(* Logix 5000 project; controller code_tcc vendor 1 type 14 code 106 rev 33.11; software revision 33.01; part 3 of 3 *)
(* tags used below, declared in another part *)
   Count : INT;
   Wrk_TransactionPtr : DINT;
(* raC_Tec_NetModbusTCPClient_ChkWrReply, continued *)

ROUTINE Prescan   (* ladder *)
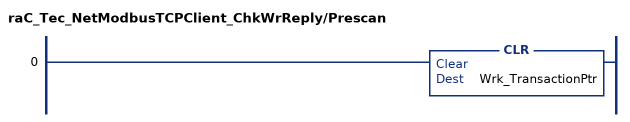
   0: CLR(Wrk_TransactionPtr);
END_ROUTINE
END_ADD_ON_INSTRUCTION

ADD_ON_INSTRUCTION raC_Tec_NetModbusTCPClient_RespStrBit   (* revision 2.0, ExecutePrescan *)
VAR_INPUT
   Inputs : BOOL; {required}
   Modbus_CMD_Len : INT; {required}
   LocalOffset : INT; {required}
END_VAR
VAR_IN_OUT
   ModbusData : raC_UDT_ModbusClientData; {required}
   CommandString : STR0500; {required}
END_VAR
VAR
   Wrk_BufferByteIndex : DINT; {access None}
   Wrk_Cmd_Last : INT; {access None}
   Wrk_Index : DINT; {access None}
   Wrk_BufferBitIndex : DINT; {access None}
   Wrk_ArraySize : DINT; {access None}
END_VAR

ROUTINE Logic   (* ladder *)
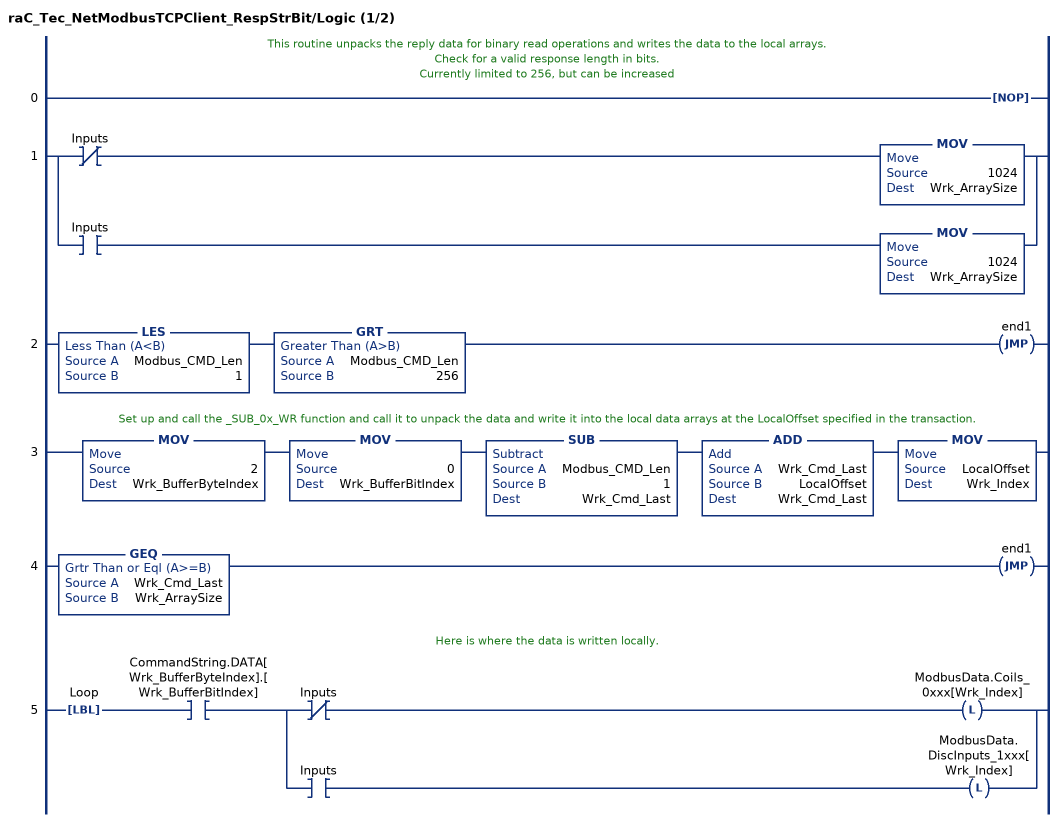
   // This routine unpacks the reply data for binary read operations and writes the data to the local arrays.
   // Check for a valid response length in bits.
   // Currently limited to 256, but can be increased
   0: NOP();
   1: [XIO(Inputs) MOV(1024,Wrk_ArraySize) ,XIC(Inputs) MOV(1024,Wrk_ArraySize) ];
   2: LES(Modbus_CMD_Len,1)GRT(Modbus_CMD_Len,256)JMP(end1);
   // Set up and call the _SUB_0x_WR function and call it to unpack the data and write it into the local data arrays at the LocalOffset specified in the transaction.
   3: MOV(2,Wrk_BufferByteIndex)MOV(0,Wrk_BufferBitIndex)SUB(Modbus_CMD_Len,1,Wrk_Cmd_Last)ADD(Wrk_Cmd_Last,LocalOffset,Wrk_Cmd_Last)MOV(LocalOffset,Wrk_Index);
   4: GEQ(Wrk_Cmd_Last,Wrk_ArraySize)JMP(end1);
   // Here is where the data is written locally.
   5: LBL(Loop)XIC(CommandString.DATA[Wrk_BufferByteIndex].[Wrk_BufferBitIndex])[XIO(Inputs) OTL(ModbusData.Coils_0xxx[Wrk_Index]) ,XIC(Inputs) OTL(ModbusData.DiscInputs_1xxx[Wrk_Index]) ];
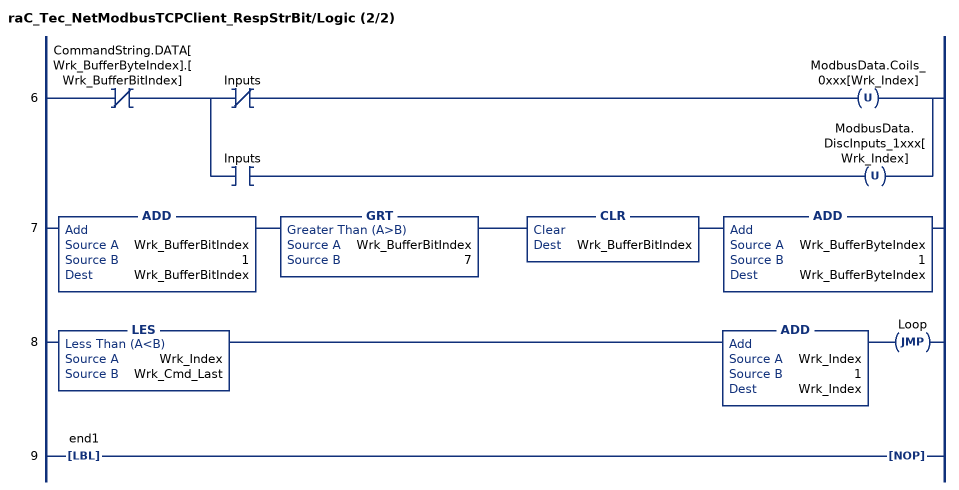
   6: XIO(CommandString.DATA[Wrk_BufferByteIndex].[Wrk_BufferBitIndex])[XIO(Inputs) OTU(ModbusData.Coils_0xxx[Wrk_Index]) ,XIC(Inputs) OTU(ModbusData.DiscInputs_1xxx[Wrk_Index]) ];
   7: ADD(Wrk_BufferBitIndex,1,Wrk_BufferBitIndex)GRT(Wrk_BufferBitIndex,7)CLR(Wrk_BufferBitIndex)ADD(Wrk_BufferByteIndex,1,Wrk_BufferByteIndex);
   8: LES(Wrk_Index,Wrk_Cmd_Last)ADD(Wrk_Index,1,Wrk_Index)JMP(Loop);
   9: LBL(end1)NOP();
END_ROUTINE

ROUTINE Prescan   (* ladder *)
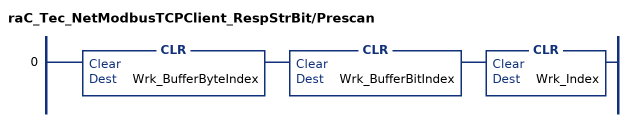
   0: CLR(Wrk_BufferByteIndex)CLR(Wrk_BufferBitIndex)CLR(Wrk_Index);
END_ROUTINE
END_ADD_ON_INSTRUCTION

ADD_ON_INSTRUCTION raC_Tec_NetModbusTCPClient_RespStrWord   (* revision 2.0, ExecutePrescan *)
VAR_INPUT
   Reg3xx : BOOL; {required}
   Modbus_CMD_Len : INT; {required}
   LocalOffset : INT; {required}
END_VAR
VAR_IN_OUT
   ModbusData : raC_UDT_ModbusClientData; {required}
   CommandString : STR0500; {required}
END_VAR
VAR
   Wrk_StringPosition : DINT; {access None}
   Wrk_Cmd_Last : INT; {access None}
   Wrk_Temp_Int : INT; {access None}
   Wrk_Index : DINT; {access None}
END_VAR

ROUTINE Logic   (* ladder *)
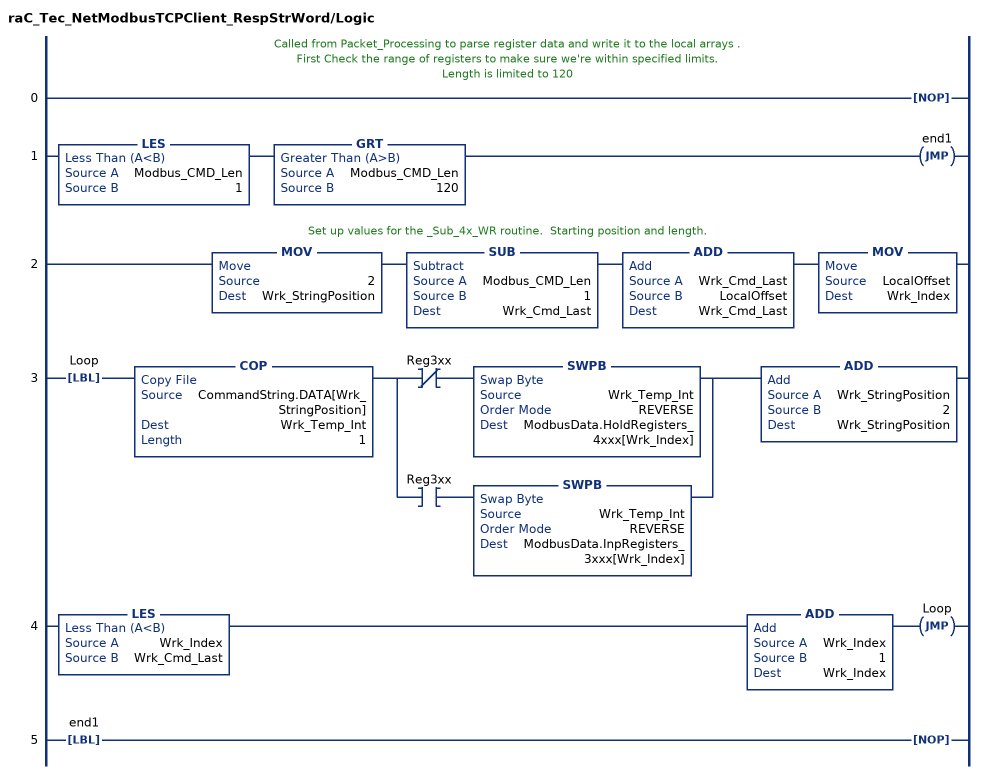
   // Called from Packet_Processing to parse register data and write it to the local arrays .
   // First Check the range of registers to make sure we're within specified limits.
   // Length is limited to 120
   0: NOP();
   1: LES(Modbus_CMD_Len,1)GRT(Modbus_CMD_Len,120)JMP(end1);
   // Set up values for the _Sub_4x_WR routine.  Starting position and length.
   2: MOV(2,Wrk_StringPosition)SUB(Modbus_CMD_Len,1,Wrk_Cmd_Last)ADD(Wrk_Cmd_Last,LocalOffset,Wrk_Cmd_Last)MOV(LocalOffset,Wrk_Index);
   3: LBL(Loop)COP(CommandString.DATA[Wrk_StringPosition],Wrk_Temp_Int,1)[XIO(Reg3xx) SWPB(Wrk_Temp_Int,REVERSE,ModbusData.HoldRegisters_4xxx[Wrk_Index]) ,XIC(Reg3xx) SWPB(Wrk_Temp_Int,REVERSE,ModbusData.InpRegisters_3xxx[Wrk_Index]) ]ADD(Wrk_StringPosition,2,Wrk_StringPosition);
   4: LES(Wrk_Index,Wrk_Cmd_Last)ADD(Wrk_Index,1,Wrk_Index)JMP(Loop);
   5: LBL(end1)NOP();
END_ROUTINE

ROUTINE Prescan   (* ladder *)
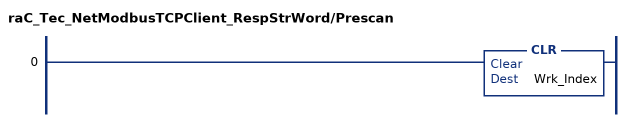
   0: CLR(Wrk_Index);
END_ROUTINE
END_ADD_ON_INSTRUCTION

VAR_GLOBAL   (* controller tags *)
   CB1_BMP : BOOL := 1;
   Client_01 : raC_Opr_NetModbusTCPClient := (Inp_Enable := 1, Sts_EN := 1, Sts_Connected := 1, Sts_Overlap := 1);
   Client_01_Data : raC_UDT_ModbusClientData := (Coils_0xxx[0] := 1, Coils_0xxx[3] := 1, Coils_0xxx[6] := 1, Coils_0xxx[10] := 1, Coils_0xxx[19] := 1, DiscInputs_1xxx[0] := 1, DiscInputs_1xxx[3] := 1, DiscInputs_1xxx[6] := 1, DiscInputs_1xxx[8] := 1, DiscInputs_1xxx[10] := 1, DiscInputs_1xxx[19] := 1);
   Client_01_EN : BOOL := 1;
   Client_01_MSG_Connect : MESSAGE;
        MessageParameters(ServiceCode := 16#004c, LocalElement := Client_01_Parameters.MSG_Src[0], ...)
   Client_01_MSG_Create : MESSAGE;
        MessageParameters(ServiceCode := 16#004b, LocalElement := Client_01_Parameters.MSG_Src[0], DestinationTag := Client_01_Parameters.MSG_Dest[0], ...)
   Client_01_MSG_Delete : MESSAGE;
        MessageParameters(ServiceCode := 16#004f, ...)
   Client_01_MSG_Read : MESSAGE;
        MessageParameters(ServiceCode := 16#004d, LocalElement := Client_01_Parameters.MSG_Src[0], DestinationTag := Client_01_Parameters.MSG_Dest[0], ...)
   Client_01_MSG_SetSing : MESSAGE;
        MessageParameters(ServiceCode := 16#0010, LocalElement := Client_01_Parameters.MSG_Src[496], ...)
   Client_01_MSG_Write : MESSAGE;
        MessageParameters(ServiceCode := 16#004e, LocalElement := Client_01_Parameters.MSG_Src[0], DestinationTag := Client_01_Parameters.MSG_Dest[0], ...)
   Client_01_Parameters : raC_UDT_ModbusClientConnection := (DestAddress := '192.168.0.10', DestinationPort := 1502, MSG_Src[0] := 20, MSG_Src[12] := 16, MSG_Src[16] := 61, MSG_Src[17] := -62, MSG_Src[21] := 10, MSG_Src[23] := 15, MSG_Src[27] := 24, MSG_Src[28] := 3, MSG_Src[29] := 73, MSG_Src[30] := 4, MSG_Src[31] := 8, MSG_Src[496] := 1, MSG_Dest[0] := 16, MSG_Dest[8] := 12, MSG_Dest[12] := 61, MSG_Dest[13] := -63, MSG_Dest[17] := 6, MSG_Dest[19] := 2, MSG_Dest[20] := 3, MSG_Dest[21] := 73, MSG_Dest[22] := 5, MSG_Dest[23] := 8, MSG_Dest[24] := 56, MSG_Dest[25] := 104, MSG_Dest[29] := 6, MSG_Dest[31] := 2, MSG_Dest[32] := 3, MSG_Dest[33] := 73, MSG_Dest[34] := 5, MSG_Dest[35] := 8, MSG_Dest[232] := 105, MSG_Dest[233] := 29, MSG_Dest[237] := 6, MSG_Dest[239] := 6);
   Client_01_Transactions : raC_UDT_ModbusClientTransaction[5] := ([0].Enabled := 1, [0].PollInterval := 80, [0].TransType := 15, [0].Count := 24, [0].TransStat := 1, [0].Diagnostic.Request := '=$C0$00$00$00$0A$00$0F$00$00$00$18$03I$04$08', [0].Diagnostic.ReqBuilt := 1, [0].Diagnostic.Overlap := 1, [0].Diagnostic.TransID := 15808, [0].Diagnostic.IntervalTimer.PRE := 40, [0].Diagnostic.IntervalTimer.ACC := 30, [0].Diagnostic.IntervalTimer.EN := 1, [0].Diagnostic.IntervalTimer.TT := 1, [0].Diagnostic.NoReplyCounter.PRE := 10, [0].Diagnostic.PendingTimer.PRE := 3000, [0].Diagnostic.PendingTimer.ACC := 110, [0].Diagnostic.PendingTimer.EN := 1, [0].Diagnostic.PendingTimer.TT := 1, [1].Enabled := 1, [1].PollInterval := 80, [1].TransType := 2, [1].Count := 24, [1].TransStat := 1, [1].Diagnostic.Request := '=$C1$00$00$00$06$00$02$00$00$00$18', [1].Diagnostic.ReqBuilt := 1, [1].Diagnostic.TransID := 15809, [1].Diagnostic.IntervalTimer.PRE := 40, [1].Diagnostic.IntervalTimer.ACC := 30, [1].Diagnostic.IntervalTimer.EN := 1, [1].Diagnostic.IntervalTimer.TT := 1, [1].Diagnostic.NoReplyCounter.PRE := 10, [1].Diagnostic.PendingTimer.PRE := 3000, [1].Diagnostic.PendingTimer.ACC := 20, [1].Diagnostic.PendingTimer.EN := 1, [1].Diagnostic.PendingTimer.TT := 1, [2].PollInterval := 1000, [2].Diagnostic.IntervalTimer.PRE := 960, [2].Diagnostic.IntervalTimer.ACC := 960, [2].Diagnostic.IntervalTimer.EN := 1, [2].Diagnostic.IntervalTimer.DN := 1, [2].Diagnostic.NoReplyCounter.DN := 1, [3].PollInterval := 1000, [3].Diagnostic.IntervalTimer.PRE := 960, [3].Diagnostic.IntervalTimer.ACC := 960, [3].Diagnostic.IntervalTimer.EN := 1, [3].Diagnostic.IntervalTimer.DN := 1, [3].Diagnostic.NoReplyCounter.DN := 1, [4].PollInterval := 1000, [4].Diagnostic.IntervalTimer.PRE := 960, [4].Diagnostic.IntervalTimer.ACC := 960, [4].Diagnostic.IntervalTimer.EN := 1, [4].Diagnostic.IntervalTimer.DN := 1, [4].Diagnostic.NoReplyCounter.DN := 1);
   contador_run : COUNTER := (PRE := 200);
   DS1_BMP : BOOL := 1;
   DS1_P1MM : BOOL := 1;
   DS1_P1MP : BOOL;
   DS1_P1WP : BOOL;
   Estado0 : BOOL := 1;
   Estado1 : BOOL;
   PM1_BMP : BOOL := 1;
   PM1_MOP : BOOL;
   PM1_MRD : BOOL;
   PM1_PMM : BOOL;
   PM1_PMP : BOOL;
   PM1_PSM : BOOL;
   PM1_PSP : BOOL;
   PM1_state : DINT;   // estados PM1: 0 = esteira rodando 1 = esteira parada e posiciona perfurador 2 = perfurador na posição e aciona perfuração 3 = perfuracao completa, comanda retorno e manda esteira p frente 0 = retorno completo volta p 0
   PM1_WPS : BOOL;
   SF1_FDM : BOOL := 1;
   SF1_FDM_TON : FBD_TIMER := (PRE := 3000);
   SF1_FDS : BOOL := 1;
   SF1_WPS : BOOL;
   teste_coil : BOOL;
   teste_var : BOOL := 1;
   ton_teste : TIMER := (PRE := 200000);
   TON_viraEsteira : TIMER := (PRE := 10000);
   TON_viraEsteira2 : TIMER := (PRE := 10000);
END_VAR

PROGRAM MainProgram   (* main routine MainRoutine *)

ROUTINE MainRoutine   (* ladder *)
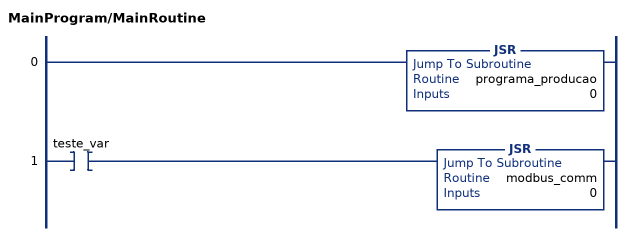
   0: JSR(programa_producao,0);
   1: XIC(teste_var)JSR(modbus_comm,0);
END_ROUTINE

ROUTINE modbus_comm   (* ladder *)
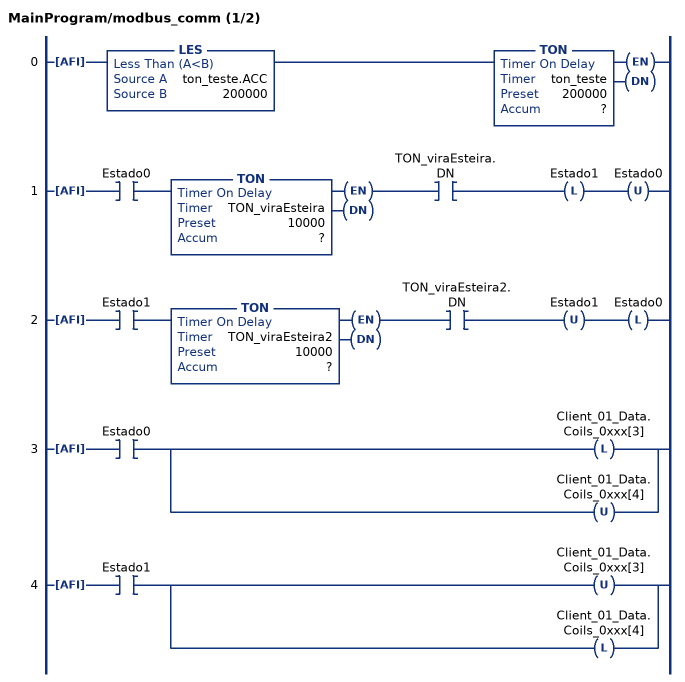
   0: AFI()LES(ton_teste.ACC,200000)TON(ton_teste,?,?);
   1: AFI()XIC(Estado0)TON(TON_viraEsteira,?,?)XIC(TON_viraEsteira.DN)OTL(Estado1)OTU(Estado0);
   2: AFI()XIC(Estado1)TON(TON_viraEsteira2,?,?)XIC(TON_viraEsteira2.DN)OTU(Estado1)OTL(Estado0);
   3: AFI()XIC(Estado0)[OTL(Client_01_Data.Coils_0xxx[3]) ,OTU(Client_01_Data.Coils_0xxx[4]) ];
   4: AFI()XIC(Estado1)[OTU(Client_01_Data.Coils_0xxx[3]) ,OTL(Client_01_Data.Coils_0xxx[4]) ];
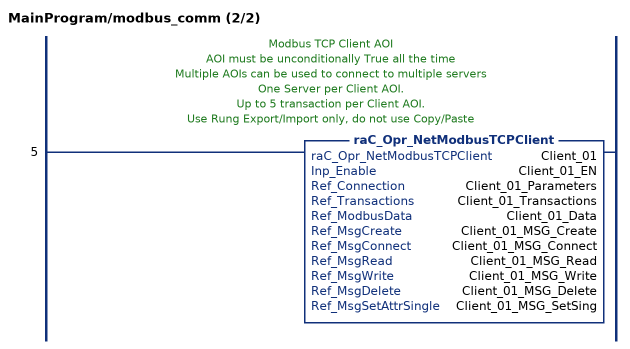
   // Modbus TCP Client AOI
   // AOI must be unconditionally True all the time
   // Multiple AOIs can be used to connect to multiple servers
   // One Server per Client AOI.
   //  Up to 5 transaction per Client AOI.
   // Use Rung Export/Import only, do not use Copy/Paste
   5: raC_Opr_NetModbusTCPClient(Client_01,Client_01_EN,Client_01_Parameters,Client_01_Transactions,Client_01_Data,Client_01_MSG_Create,Client_01_MSG_Connect,Client_01_MSG_Read,Client_01_MSG_Write,Client_01_MSG_Delete,Client_01_MSG_SetSing);
END_ROUTINE

ROUTINE programa_producao   (* structured text *)
   DS1_P1WP := Client_01_Data.DiscInputs_1xxx[9];
   PM1_MRD := Client_01_Data.DiscInputs_1xxx[13];
   PM1_PSP := Client_01_Data.DiscInputs_1xxx[16];
   PM1_PSM := Client_01_Data.DiscInputs_1xxx[17];
   PM1_WPS := Client_01_Data.DiscInputs_1xxx[18];
   SF1_WPS := Client_01_Data.DiscInputs_1xxx[21];
   SF1_FDS := Client_01_Data.DiscInputs_1xxx[20];
   
   /*IF SF1_WPS AND SF1_FDS THEN
   	SF1_FDM := 1;
   end_if;
   SF1_FDM_TON.PRE := 3000;
   SF1_FDM_TON.TimerEnable := SF1_FDM;
   TONR(SF1_FDM_TON);
   IF SF1_FDM_TON.DN then
   	SF1_FDM := 0;
   	SF1_FDM_TON.Reset := 1;
   else
   	SF1_FDM_TON.Reset := 0;
   end_if;*/
   SF1_FDM := 1;
   
   //PM1:
   /*
   estados PM1:
   
   0 = esteira rodando
   1 = esteira parada e posiciona perfurador
   2 = perfurador na posição e aciona perfuração
   3 = perfuracao completa, comanda retorno e manda esteira p frente
   0 = retorno completo volta p 0
   */
   //PM1 transições de estado
   IF NOT PM1_WPS AND NOT PM1_PSM AND PM1_state <> 1 AND PM1_state <> 2 then
   	PM1_state := 0;
   	PM1_PMM := 0;
   end_if;
   IF PM1_WPS AND PM1_state = 0 then
   	PM1_state := 1;
   end_if;
   IF PM1_state = 1 AND PM1_PSP AND PM1_PSM AND PM1_MRD then
   	PM1_state := 2;
   end_if;
   IF NOT PM1_MRD AND PM1_state = 2 THEN
   	PM1_state := 3;
   end_if;
   
   //ações
   IF PM1_state = 0 then
   	PM1_BMP := 1; // manda esteira p frente
   end_if;
   IF PM1_state = 1 then
   	PM1_BMP := 0; // para esteira
   	PM1_PMP := 1; // posiciona furador
   end_if;
   IF PM1_state = 2 then
   	PM1_MOP := 1; // manda perfurar
   end_if;
   IF PM1_state = 3 then
   	PM1_MOP := 0; // desliga perfuração
   	PM1_PMP := 0; // para comando de posicionamento
   	PM1_PMM := 1; // comanda p retornar perfurador
   	PM1_BMP := 1; // manda esteira p frente
   end_if;
   
   CB1_BMP := 1;
   
   DS1_BMP :=1;
   DS1_P1MM := 1;
   DS1_P1MP := 0;
   IF DS1_P1WP then
   	DS1_BMP := 0;
   	DS1_P1MM := 0;
   	DS1_P1MP := 1;
   end_if;
   
   // mapeamento de variaveis
   
   Client_01_Data.Coils_0xxx[0] := CB1_BMP;
   Client_01_Data.Coils_0xxx[3] := DS1_BMP;
   Client_01_Data.Coils_0xxx[5] := DS1_P1MP;
   Client_01_Data.Coils_0xxx[6] := DS1_P1MM;
   Client_01_Data.Coils_0xxx[10] := PM1_BMP;
   Client_01_Data.Coils_0xxx[12] := PM1_MOP;
   Client_01_Data.Coils_0xxx[14] := PM1_PMP;
   Client_01_Data.Coils_0xxx[15] := PM1_PMM;
   Client_01_Data.Coils_0xxx[19] := SF1_FDM;
END_ROUTINE
END_PROGRAM
